FUNCTION_BLOCK FB_MotorsPowerUp
VAR_INPUT
	bExecute : BOOL;
END_VAR
VAR_OUTPUT
	bPowerUpError 	: BOOL := FALSE;
	bPowerUpDone 	: BOOL := FALSE;
END_VAR
VAR
	eState    	: (Reset, M1, M2, M3, M4, M5, M6, M7, M8); 
	fbMCPowerM1, fbMCPowerM2, fbMCPowerM3, fbMCPowerM4, fbMCPowerM5, fbMCPowerM6, fbMCPowerM7, fbMCPowerM8	: FB_MCPower;
		PowerErrorID	: UDINT;
		bPowerStatus	: BOOL := FALSE;
		bM2 : BOOL := FALSE;
		bM3 : BOOL := FALSE;
END_VAR

CASE eState OF
	Reset:
		bPowerUpDone := FALSE;
		eState := M1;
	M1:
		IF bExecute THEN
			fbMcPowerM1(
				Axis 			:= GVL_Motion.M1Motor.Axis,	//axisPointer^,
				bEnable 		:= TRUE, 	//Enable the Axis if the driver is ready without safety fauls
				bError			=> bPowerUpError,
				iErrorID		=> PowerErrorID,	 //Error ID if the power enter in error.
				bActive			=> bPowerStatus
			);
		END_IF
		IF fbMCPowerM1.bActive THEN
			eState := M2;
			//bPowerUpDone := TRUE;
		END_IF
	M2:
		IF bExecute THEN
			fbMcPowerM2(
				Axis 			:= GVL_Motion.M2Motor.Axis,	//axisPointer^,
				bEnable 		:= TRUE, 	//Enable the Axis if the driver is ready without safety fauls
				bError			=> bPowerUpError,
				iErrorID		=> PowerErrorID,	 //Error ID if the power enter in error.
				bActive			=> bPowerStatus
			);
		END_IF
		IF fbMCPowerM2.bActive THEN
			eState := M3;
			//bPowerUpDone := TRUE;
		END_IF
	
	M3:
		IF bExecute THEN
			fbMcPowerM3(
				Axis 			:= GVL_Motion.M3Motor.Axis,	//axisPointer^,
				bEnable 		:= TRUE, 	//Enable the Axis if the driver is ready without safety fauls
				bError			=> bPowerUpError,
				iErrorID		=> PowerErrorID,	 //Error ID if the power enter in error.
				bActive			=> bPowerStatus
			);
		END_IF
		IF fbMCPowerM3.bActive THEN
			eState := M4;
			//bPowerUpDone := TRUE;
		END_IF
		
	M4: //VICI Valve 1
		IF bExecute THEN
			fbMcPowerM4(
				Axis 			:= GVL_Motion.aValves[1].Axis,	//axisPointer^,
				bEnable 		:= TRUE, 	//Enable the Axis if the driver is ready without safety fauls
				bError			=> bPowerUpError,
				iErrorID		=> PowerErrorID,	 //Error ID if the power enter in error.
				bActive			=> bPowerStatus
			);
		END_IF
		IF fbMCPowerM4.bActive THEN
			eState := M5;
			//bPowerUpDone := TRUE;
		END_IF
		
	M5: //VICI Valve 2
		IF bExecute THEN
			fbMcPowerM5(
				Axis 			:= GVL_Motion.aValves[2].Axis,	//axisPointer^,
				bEnable 		:= TRUE, 	//Enable the Axis if the driver is ready without safety fauls
				bError			=> bPowerUpError,
				iErrorID		=> PowerErrorID,	 //Error ID if the power enter in error.
				bActive			=> bPowerStatus
			);
		END_IF
		IF fbMCPowerM5.bActive THEN
			eState := M6;
			//bPowerUpDone := TRUE;
		END_IF
		
	M6: //VICI Valve 3
		IF bExecute THEN
			fbMcPowerM6(
				Axis 			:= GVL_Motion.aValves[3].Axis,	//axisPointer^,
				bEnable 		:= TRUE, 	//Enable the Axis if the driver is ready without safety fauls
				bError			=> bPowerUpError,
				iErrorID		=> PowerErrorID,	 //Error ID if the power enter in error.
				bActive			=> bPowerStatus
			);
		END_IF
		IF fbMCPowerM6.bActive THEN
			eState := M7;
			//bPowerUpDone := TRUE;
		END_IF
		
	M7: //VICI Valve 4
		IF bExecute THEN
			fbMcPowerM7(
				Axis 			:= GVL_Motion.aValves[4].Axis,	//axisPointer^,
				bEnable 		:= TRUE, 	//Enable the Axis if the driver is ready without safety fauls
				bError			=> bPowerUpError,
				iErrorID		=> PowerErrorID,	 //Error ID if the power enter in error.
				bActive			=> bPowerStatus
			);
		END_IF
		IF fbMCPowerM7.bActive THEN
			eState := M8;
			//bPowerUpDone := TRUE;
		END_IF
		 
	M8: //VICI Valve 5
		IF bExecute THEN
			fbMcPowerM8(
				Axis 			:= GVL_Motion.aValves[5].Axis,	//axisPointer^,
				bEnable 		:= TRUE, 	//Enable the Axis if the driver is ready without safety fauls
				bError			=> bPowerUpError,
				iErrorID		=> PowerErrorID,	 //Error ID if the power enter in error.
				bActive			=> bPowerStatus
			);
		END_IF
		IF fbMCPowerM8.bActive THEN
			bPowerUpDone := TRUE;
		END_IF
	
END_CASE

END_FUNCTION_BLOCK

(* stored: Version 1.1.0.1, ProductVersion 3.1.4024.12
   POU FB_MotorsPowerUp: Id {2ede40b4-9170-4e3a-965e-058f9fe9c946}, SpecialFunc None *)
